FUNCTION_BLOCK FB_HMI_TILT_A EXTENDS FB_HMI_COMPONENT
VAR_OUTPUT
END_VAR
VAR_IN_OUT
    fbInstance : FB_NOTT_TIP_TILT;
END_VAR
VAR
END_VAR

fbHealthStatus(

    bIsGood := NOT fbInstance.stat.bError,
    bHasWarning := (    fbInstance.stat.bWarning));
                     
fbBusyStatus(
    bIsBusy := FALSE);

M_UpdateStatusColor();

END_FUNCTION_BLOCK

(* stored: Version 1.1.0.1, ProductVersion 3.1.4024.14
   POU FB_HMI_TILT_A: Id {0b16a9cd-e0ad-4543-be57-a37398cc6741}, SpecialFunc None *)
